// TIA Portal V17 export
// export: Created 2025-03-07T09:19:50.7944546Z, ExportSetting WithDefaults, DisplayName Totally Integrated Automation Portal, DisplayVersion V17 Update 8, DisplayName TIA Portal Openness, DisplayVersion V17 Update 8, DisplayName TIA Portal Version Control Interface, DisplayVersion V17, DisplayName SINAMICS Startdrive Advanced, DisplayVersion V17 SP2, DisplayName SINAMICS Startdrive G110M, G120, G120C, G120D, G120P, G115D, DisplayVersion V17 SP2, DisplayName SINAMICS Startdrive G130, G150, S120, S150, SINAMICS MV, S210, DisplayVersion V17 SP2, DisplayName STEP 7 Professional, DisplayVersion V17 Update 8, DisplayName SINUMERIK ONE STEP 7 Toolbox, DisplayVersion V17 Update 12, DisplayName SINUMERIK 840D sl STEP 7 Toolbox, DisplayVersion V17 Update 12, DisplayName STEP 7 Safety, DisplayVersion V17 Update 6, DisplayName WinCC Advanced, DisplayVersion V17 Update 8
TYPE "ADVANCE_RETURN_CYL_CLADDING"
// stored: IsFailsafeCompliant false
   STRUCT
      GENERAL_CONDITIONS : Bool;   // GENERAL CONDITIONS
      ADVANCE_CONDITIONS : Bool;   // ADVANCE CONDITIONS
      RETURN_CONDITIONS : Bool;   // RETURN CONDITIONS
      GENERAL_CONDITIONS_HELP : Bool;   // GENERAL CONDITIONS HELP
      ADVANCE_CONDITIONS_HELP : Bool;   // ADVANCE CONDITIONS HELP
      RETURN_CONDITIONS_HELP : Bool;   // RETURN CONDITIONS HELP
      ADVANCE_HMI_REQUEST : Bool;   // ADVANCE HMI REQUEST / ADVANCE MANUAL HMI REQUEST
      RETURN_HMI_REQUEST : Bool;   // RETURN HMI REQUEST / RETURN MANUAL HMI REQUEST
      ADVANCE_MANUAL_REQUEST : Bool;   // ADVANCE MANUAL REQUEST
      RETURN_MANUAL_REQUEST : Bool;   // RETURN MANUAL REQUEST
      ADVANCE_AUTO_REQUEST : Bool;   // ADVANCE AUTO REQUEST
      RETURN_AUTO_REQUEST : Bool;   // RETURN AUTO REQUEST
      ADVANCE_GLOBAL_REQUEST : Bool;   // ADVANCE GLOBAL REQUEST
      RETURN_GLOBAL_REQUEST : Bool;   // RETURN GLOBAL REQUEST
      ADVANCE_COMMAND : Bool;   // ADVANCE COMMAND
      RETURN_COMMAND : Bool;   // RETURN COMMAND
      FULL_ADVANCED : Bool;   // ADVANCED FEEDBACK / ADVANCED AND COMMANDED
      FULL_RETURNED : Bool;   // RETURNED FEEDBACK / RETURNED AND COMMANDED
      SIMULTANEITY_ALARM : Bool;   // SIMULTANEITY FAULT / SIMULTANEITY ALARM
      TIME_EXCEEDED_ALARM : Bool;   // TIME EXCEEDED / TIME EXCEEDED ALARM
      ANY_ACTIVE_ALARM : Bool;   // FAULT / ANY ACTIVE ALARM
      IS_SEOC_ALARMS : Bool;   // INMEDIATE STOP AND STOP END OF CYCLE ALARMS
      PULSE_1 : Bool;   // PULSE 1
      PULSE_2 : Bool;   // PULSE 2
      PULSE_3 : Bool;   // PULSE 3
   END_STRUCT;
END_TYPE
